{attribute 'qualified_only'}
{attribute 'strict'}
TYPE ENUM_LaserCoupling_States :
(
    Unknown := 0,
    OUT := 1,
    Mirror1 := 2

)UINT;
END_TYPE

(* stored: Version 1.1.0.1, ProductVersion 3.1.4022.18
   DUT ENUM_LaserCoupling_States: Id {3ae742f5-a942-463c-843b-aed92c25891d} *)
